INTERFACE I_EventBase

METHOD Clear : BOOL
VAR_INPUT
END_VAR
END_METHOD

METHOD ClearAllEvents : HRESULT
VAR_INPUT
END_VAR
END_METHOD

METHOD Confirm : HRESULT
VAR_INPUT
END_VAR
END_METHOD

METHOD Create : HRESULT
VAR_INPUT
END_VAR
END_METHOD

METHOD Raise : HRESULT
VAR_INPUT
END_VAR
END_METHOD

END_INTERFACE

(* stored: Version 1.1.0.1, ProductVersion 3.1.4024.14
   Itf I_EventBase: Id {5e78eace-093f-43b4-9a3c-92dc170144de}
   Method Clear: Id {b0b2854d-9854-4b39-826f-5f9f2e3e706a}
   Method ClearAllEvents: Id {9e60c04a-1a60-464a-b40f-f78409187b2f}
   Method Confirm: Id {8030da31-0c7b-41e3-8f25-4700077e9568}
   Method Create: Id {f3b622be-6e0e-4718-865a-ad8f829fe210}
   Method Raise: Id {4c4af0e7-a4bd-4446-a127-69fa8c2edefc} *)
